(* Logix 5000 project; controller RSL5k_18_Template_noLib Emulate 5570 rev 32.11; software revision 32.02; part 2 of 16 *)
(* tags used below, declared in another part *)
   Inp_PV : REAL;   // Input Signal (process variable) from Sensor
   Inp_PVSrcQ : DINT;   // Input Source and Quality (from Channel object, if available) (enum)
   Inp_PVNotify : DINT;   // Related PV object alarm prio and ack status (enum)
   Inp_PVBad : BOOL;   // 1=PV or I/O Comms Status Bad, 0=OK
   Inp_PVUncertain : BOOL;   // 1=PV Value Not Reliable, 0=OK
   Inp_Sim : BOOL;   // 1=Use simulated PV (Set_SimPV); 0=Use Input (Inp_PV)
   Cfg_UseChanSrcQ : BOOL;   // 1=Pass thru connected Channel's SrcQ value, 0=generate SrcQ
   Cfg_FiltTC : REAL;   // PV Filter Time Constant (s), 0.0 = unfiltered
   Cfg_HiHiLim : REAL;   // High-High Status Threshold (EU)
   Cfg_HiHiDB : REAL;   // High-High Status Deadband (EU)
   Cfg_HiLim : REAL;   // High Status Threshold (EU)
   Cfg_HiDB : REAL;   // High Status Deadband (EU)
   Cfg_LoLim : REAL;   // Low Status Threshold (EU)
   Cfg_LoDB : REAL;   // Low Status Deadband (EU)
   Cfg_LoLoLim : REAL;   // Low-Low Status Threshold (EU)
   Cfg_LoLoDB : REAL;   // Low-Low Status Deadband (EU)
   Cfg_FailHiLim : REAL;   // Out-of-Range (fail) High Limit (raw units)
   Cfg_FailLoLim : REAL;   // Out-of-Range (fail) Low Limit (raw units)
   Cfg_FailDB : REAL;   // Out-of-Range (fail) High/Low Deadband (raw units)
   Set_SimPV : REAL;   // PV used in Simulation (Inp_Sim=1) (EU)
   PCmd_ClearCapt : BOOL;   // Program Command to Clear the captured min / max PV excursion values
   Val : REAL;   // Analog Value (after Substitute PV, if used)
   Val_InpPV : REAL;   // Analog Input Value (actual, before Substitute PV selection)
   Val_PVMinCapt : REAL;   // Captured PV Minimum (excursion) since last cleared
   Val_PVMaxCapt : REAL;   // Captured PV Maximum (excursion) since last cleared
   SrcQ_IO : DINT;   // Source and Quality of primary I/O (enumeration)
   SrcQ : DINT;   // Source and Quality of primary Val/Sts (enumeration)
   Val_Fault : DINT;   // Device Fault Status 0=none, 20=Lo, 21=Hi, 24=LoLo, 25=HiHi, 32=Fail, 34=CfgErr
   Val_NotifyAll : DINT;   // Highest Alarm prio and ack status this object + channel (enum)
   Val_UnackAlmC : DINT;   // Count of Unacknowledged Alarms
   Sts_SubstPV : BOOL;   // 1=Using Substitute PV (overrides input), 0=Using live Input PV from device
   Sts_PVBad : BOOL;   // 1=PV Bad quality or Out of Range
   Sts_PVUncertain : BOOL;   // 1=PV Value is Uncertain (quality)
   Sts_AlmInh : BOOL;   // 1=An Alarm is Shelved, Disabled or Suppressed: display icon
   Sts_Err : BOOL;   // 1=Error in Config (see detail Err_ bits for reason), display icon
   Err_Raw : BOOL;   // 1=Error in Config: Raw Input Scaling Min = Max
   Err_EU : BOOL;   // 1=Error in Config: Scaled EU Min = Max
   Err_Timer : BOOL;   // 1=Error in Config: On Delay, Off Delay, Gate Delay Time Invalid (use 0 to 2147483 s)
   Err_Filt : BOOL;   // 1=Error in Config: PV filter params (RateTime, TC)
   Err_Alarm : BOOL;   // 1=Error in Config: Alarm Min On Time, Shelf Time, Severity
   Sts_RdyReset : ALIAS FOR ORdy_Reset;   // 1=A latched alarm or shed condition is ready to be reset
   Sts_RdyAck : BOOL;   // 1=An alarm is ready to be acknowledged
   Sts_HiHiCmp : ALIAS FOR HiHiGate.Inp;   // PV High-High comparison result 1=High-High
   Sts_HiHi : ALIAS FOR HiHi.Inp;   // 1=Analog Input is above High-High limit
   Sts_HiCmp : ALIAS FOR HiGate.Inp;   // PV High comparison result 1=High
   Sts_Hi : ALIAS FOR Hi.Inp;   // 1=Analog Input is above High limit
   Sts_LoCmp : ALIAS FOR LoGate.Inp;   // PV Low comparison result 1=Low
   Sts_Lo : ALIAS FOR Lo.Inp;   // 1=Analog Input is below Low limit
   Sts_LoLoCmp : ALIAS FOR LoLoGate.Inp;   // PV Low-Low comparison result 1=Low-Low
   Sts_LoLo : ALIAS FOR LoLo.Inp;   // 1=Analog Input is below Low-Low limit
   Sts_FailCmp : ALIAS FOR FailGate.Inp;   // PV Fail comparison result 1=Out of Range
   Sts_Fail : ALIAS FOR Fail.Inp;   // 1=Analog Input is Out of Range or PV Bad
   P_AIn : BOOL;   // Unique Parameter Name for auto - discovery
   LoLo : P_Alarm;   // Low-Low Alarm
   Lo : P_Alarm;   // Low Alarm
   Hi : P_Alarm;   // High Alarm
   HiHi : P_Alarm;   // High-High Alarm
   Fail : P_Alarm;   // Analog Input Failure Alarm (bad quality or out of range)
   Wrk_Notify : DINT;   // Buffer for building Val_Notify
   Wrk_Fault : DINT;   // Buffer for building Val_Fault
   Wrk_SrcQ : DINT;   // Register for building Source / Quality enumeration
   Wrk_SubstPV : BOOL;   // Internal flag: Using Substitute PV
   Wrk_UnfiltPV : REAL;   // Unfiltered PV, input to 1st order filter
   Wrk_Alpha : REAL;   // Filter multiplier = (1 / (1+TC/dT) )
   Wrk_ScanT : TIMER;   // Scan Timer (milliseconds, always runs)
   Wrk_ScanTime : REAL;   // Time since this instance was last scanned
   Wrk_FiltPV : REAL;   // Filtered PV
   Wrk_ValidONS : BOOL;   // Selected PV goes from Infinite or Not a Number to VALID
   Wrk_SelPVDINT : DINT;   // Selected PV check for Infinite or Non A Number
   Wrk_SelPVInfNaN : BOOL;   // Selected PV (Input or Substitute) is Infinite or NaN
   Wrk_Fail : BOOL;   // Internal flag: Fail Status
   Wrk_LoLo : BOOL;   // Internal flag: Low-Low Status
   Wrk_Lo : BOOL;   // Internal flag: Low Status
   Wrk_Hi : BOOL;   // Internal flag: High Status
   Wrk_HiHi : BOOL;   // Internal flag: High-High Status
   FailGate : P_Gate;   // Fail Alarm Gate / Delay Block
   LoLoGate : P_Gate;   // Low-Low Alarm Gate / Delay Block
   LoGate : P_Gate;   // Low Alarm Gate / Delay Block
   HiHiGate : P_Gate;   // High-High Alarm Gate / Delay Block
   HiGate : P_Gate;   // High Alarm Gate / Delay Block
   Wrk_InpInfNaN : BOOL;   // Input is Infinite or Not a Number
   Wrk_UnackAlmC : DINT;   // Buffer for building Val_UnackAlmC
   Val_Notify : DINT;   // Highest Alarm prio and ack status this object only (enum)
   ORdy_ResetAckAll : BOOL;   // 1=Ready for OCmd_ResetAckAll (enables HMI button)
   ORdy_Reset : BOOL;   // 1=Ready for OCmd_Reset (enables HMI button)
   OCmd_ClearCapt : BOOL;   // Operator Command to Clear the captured min / max PV excursion values
   MSet_SubstPV : REAL;   // Maintenance-Entered Substitute PV (EU)
   Wrk_RawPV : REAL;   // Value of raw PV to be used for Out of Range checking
(* P_AIn, continued *)

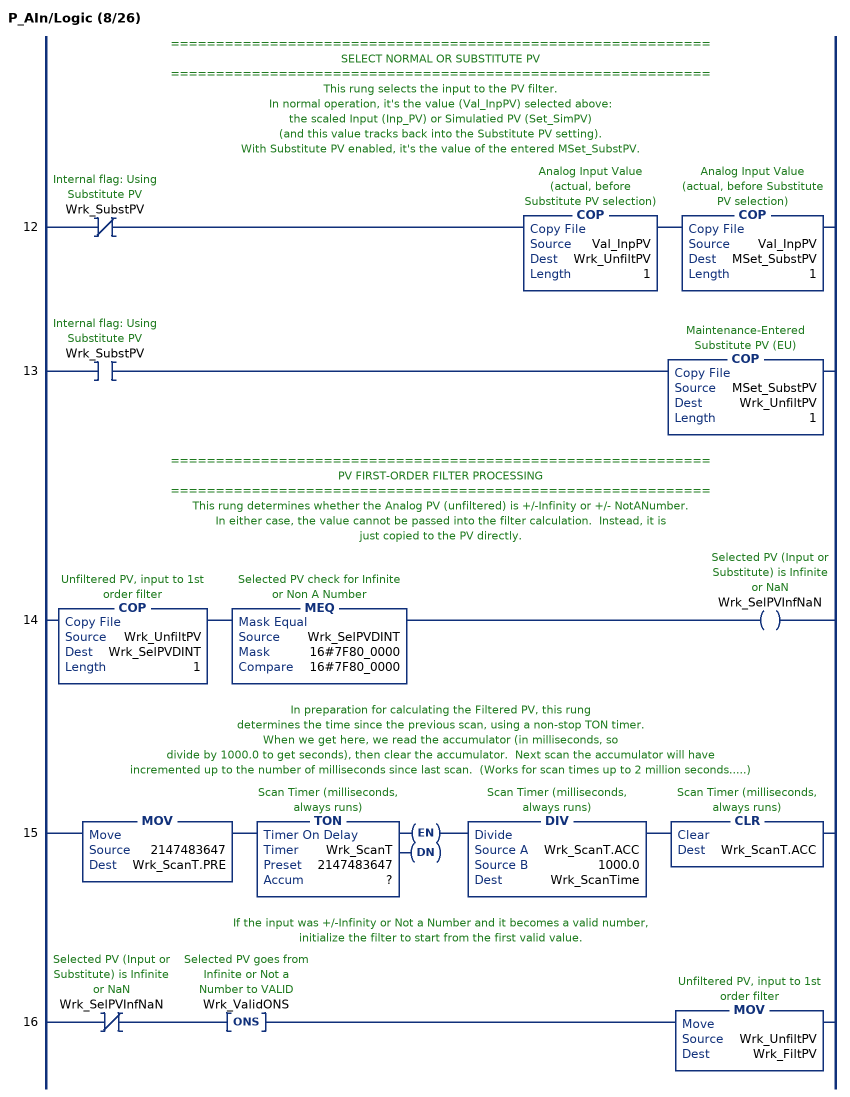
   [picture p24: P_AIn/Logic rungs 12-16]
   // ============================================================
   // SELECT NORMAL OR SUBSTITUTE PV
   // ============================================================
   // This rung selects the input to the PV filter.
   // In normal operation, it's the value (Val_InpPV) selected above:
   // the scaled Input (Inp_PV) or Simulatied PV (Set_SimPV)
   // (and this value tracks back into the Substitute PV setting).
   // With Substitute PV enabled, it's the value of the entered MSet_SubstPV.
   12: XIO(Wrk_SubstPV)COP(Val_InpPV,Wrk_UnfiltPV,1)COP(Val_InpPV,MSet_SubstPV,1);
   13: XIC(Wrk_SubstPV)COP(MSet_SubstPV,Wrk_UnfiltPV,1);
   // ============================================================
   // PV FIRST-ORDER FILTER PROCESSING
   // ============================================================
   // This rung determines whether the Analog PV (unfiltered) is +/-Infinity or +/- NotANumber.
   // In either case, the value cannot be passed into the filter calculation.  Instead, it is
   // just copied to the PV directly.
   14: COP(Wrk_UnfiltPV,Wrk_SelPVDINT,1)MEQ(Wrk_SelPVDINT,16#7F80_0000,16#7F80_0000)OTE(Wrk_SelPVInfNaN);
   // In preparation for calculating the Filtered PV, this rung
   // determines the time since the previous scan, using a non-stop TON timer.
   // When we get here, we read the accumulator (in milliseconds, so
   // divide by 1000.0 to get seconds), then clear the accumulator.  Next scan the accumulator will have
   // incremented up to the number of milliseconds since last scan.  (Works for scan times up to 2 million seconds.....)
   15: MOV(2147483647,Wrk_ScanT.PRE)TON(Wrk_ScanT,?,?)DIV(Wrk_ScanT.ACC,1000.0,Wrk_ScanTime)CLR(Wrk_ScanT.ACC);
   // If the input was +/-Infinity or Not a Number and it becomes a valid number,
   // initialize the filter to start from the first valid value.
   16: XIO(Wrk_SelPVInfNaN)ONS(Wrk_ValidONS)MOV(Wrk_UnfiltPV,Wrk_FiltPV);
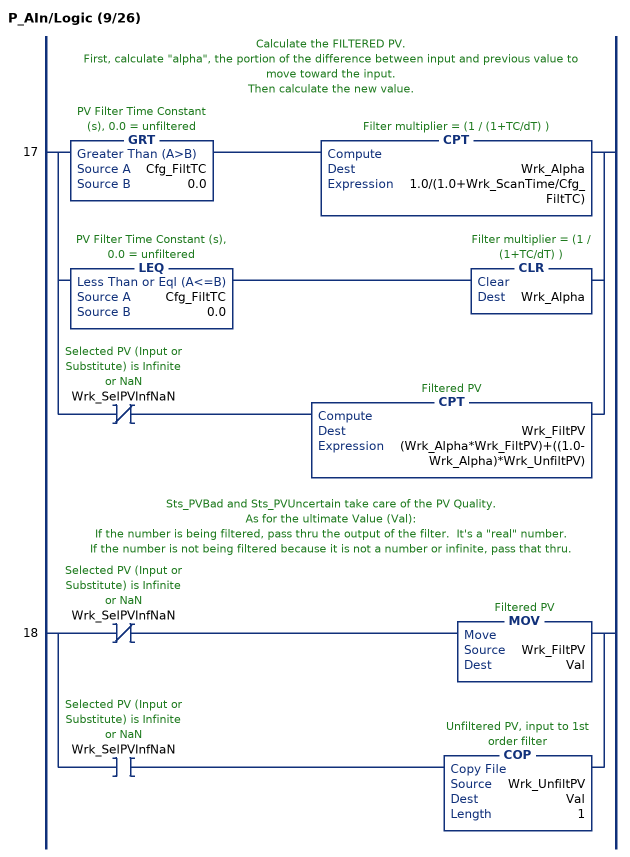
   // Calculate the FILTERED PV.
   // First, calculate "alpha", the portion of the difference between input and previous value to move toward the input.
   // Then calculate the new value.
   17: [GRT(Cfg_FiltTC,0.0) CPT(Wrk_Alpha,1.0/(1.0+Wrk_ScanTime/Cfg_FiltTC)) ,LEQ(Cfg_FiltTC,0.0) CLR(Wrk_Alpha) ,XIO(Wrk_SelPVInfNaN) CPT(Wrk_FiltPV,(Wrk_Alpha*Wrk_FiltPV)+((1.0-Wrk_Alpha)*Wrk_UnfiltPV)) ];
   // Sts_PVBad and Sts_PVUncertain take care of the PV Quality.
   // As for the ultimate Value (Val):
   // If the number is being filtered, pass thru the output of the filter.  It's a "real" number.
   // If the number is not being filtered because it is not a number or infinite, pass that thru.
   18: [XIO(Wrk_SelPVInfNaN) MOV(Wrk_FiltPV,Val) ,XIC(Wrk_SelPVInfNaN) COP(Wrk_UnfiltPV,Val,1) ];
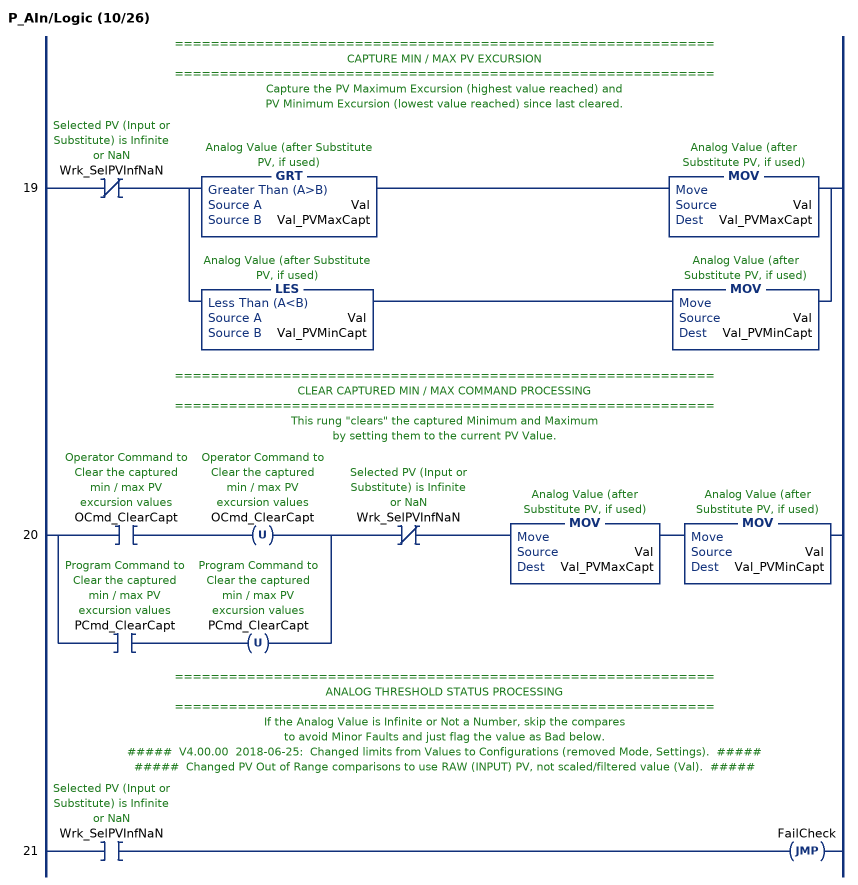
   // ============================================================
   // CAPTURE MIN / MAX PV EXCURSION
   // ============================================================
   // Capture the PV Maximum Excursion (highest value reached) and
   // PV Minimum Excursion (lowest value reached) since last cleared.
   19: XIO(Wrk_SelPVInfNaN)[GRT(Val,Val_PVMaxCapt) MOV(Val,Val_PVMaxCapt) ,LES(Val,Val_PVMinCapt) MOV(Val,Val_PVMinCapt) ];
   // ============================================================
   // CLEAR CAPTURED MIN / MAX COMMAND PROCESSING
   // ============================================================
   // This rung "clears" the captured Minimum and Maximum
   // by setting them to the current PV Value.
   20: [XIC(OCmd_ClearCapt) OTU(OCmd_ClearCapt) ,XIC(PCmd_ClearCapt) OTU(PCmd_ClearCapt) ]XIO(Wrk_SelPVInfNaN)MOV(Val,Val_PVMaxCapt)MOV(Val,Val_PVMinCapt);
   // ============================================================
   // ANALOG THRESHOLD STATUS PROCESSING
   // ============================================================
   // If the Analog Value is Infinite or Not a Number, skip the compares
   // to avoid Minor Faults and just flag the value as Bad below.
   // #####  V4.00.00  2018-06-25:  Changed limits from Values to Configurations (removed Mode, Settings).  #####
   // #####  Changed PV Out of Range comparisons to use RAW (INPUT) PV, not scaled/filtered value (Val).  #####
   21: XIC(Wrk_SelPVInfNaN)JMP(FailCheck);
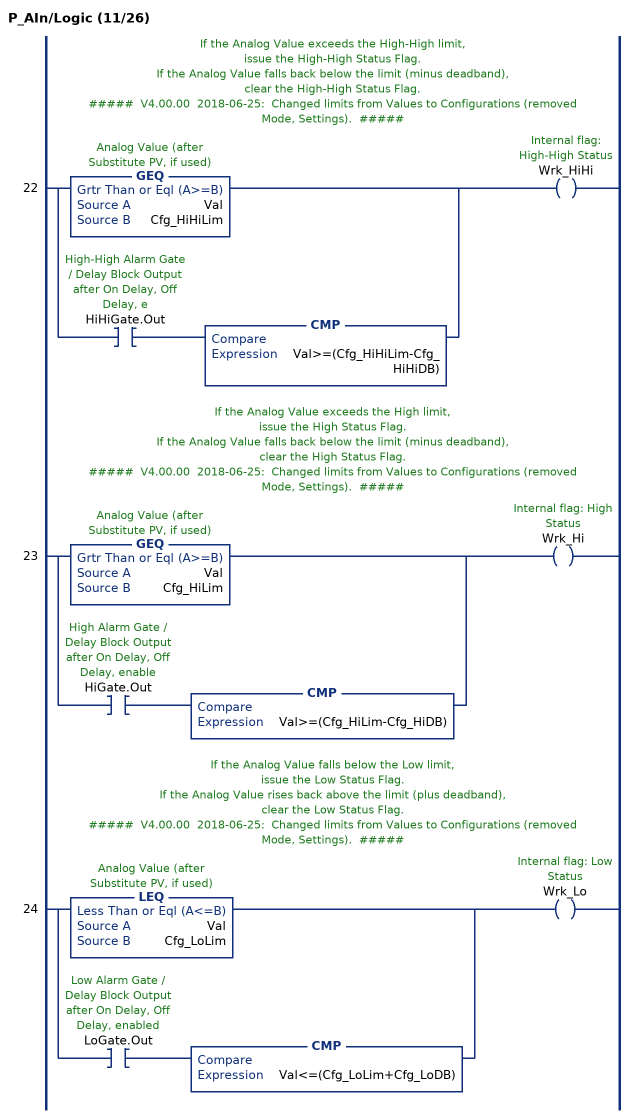
   // If the Analog Value exceeds the High-High limit,
   // issue the High-High Status Flag.
   // If the Analog Value falls back below the limit (minus deadband),
   // clear the High-High Status Flag.
   // #####  V4.00.00  2018-06-25:  Changed limits from Values to Configurations (removed Mode, Settings).  #####
   22: [GEQ(Val,Cfg_HiHiLim) ,XIC(HiHiGate.Out) CMP(Val>=(Cfg_HiHiLim-Cfg_HiHiDB)) ]OTE(Wrk_HiHi);
   // If the Analog Value exceeds the High limit,
   // issue the High Status Flag.
   // If the Analog Value falls back below the limit (minus deadband),
   // clear the High Status Flag.
   // #####  V4.00.00  2018-06-25:  Changed limits from Values to Configurations (removed Mode, Settings).  #####
   23: [GEQ(Val,Cfg_HiLim) ,XIC(HiGate.Out) CMP(Val>=(Cfg_HiLim-Cfg_HiDB)) ]OTE(Wrk_Hi);
   // If the Analog Value falls below the Low limit,
   // issue the Low Status Flag.
   // If the Analog Value rises back above the limit (plus deadband),
   // clear the Low Status Flag.
   // #####  V4.00.00  2018-06-25:  Changed limits from Values to Configurations (removed Mode, Settings).  #####
   24: [LEQ(Val,Cfg_LoLim) ,XIC(LoGate.Out) CMP(Val<=(Cfg_LoLim+Cfg_LoDB)) ]OTE(Wrk_Lo);
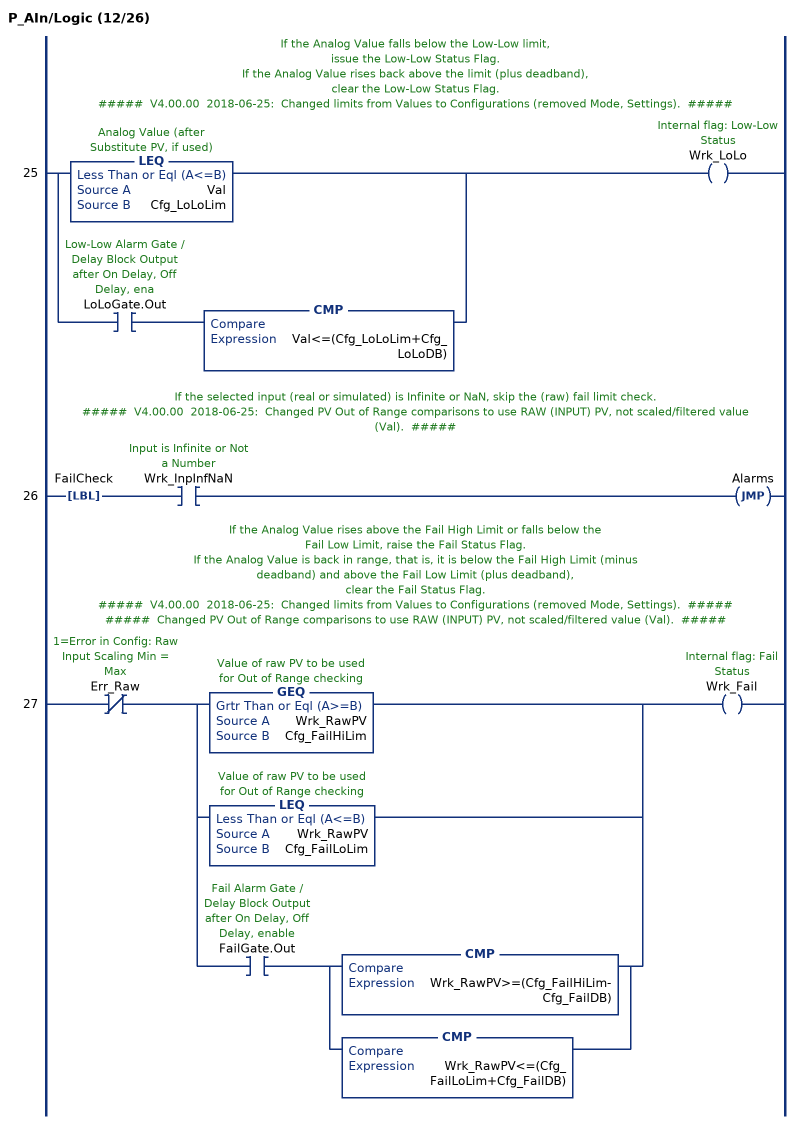
   // If the Analog Value falls below the Low-Low limit,
   // issue the Low-Low Status Flag.
   // If the Analog Value rises back above the limit (plus deadband),
   // clear the Low-Low Status Flag.
   // #####  V4.00.00  2018-06-25:  Changed limits from Values to Configurations (removed Mode, Settings).  #####
   25: [LEQ(Val,Cfg_LoLoLim) ,XIC(LoLoGate.Out) CMP(Val<=(Cfg_LoLoLim+Cfg_LoLoDB)) ]OTE(Wrk_LoLo);
   // If the selected input (real or simulated) is Infinite or NaN, skip the (raw) fail limit check.
   // #####  V4.00.00  2018-06-25:  Changed PV Out of Range comparisons to use RAW (INPUT) PV, not scaled/filtered value (Val).  #####
   26: LBL(FailCheck)XIC(Wrk_InpInfNaN)JMP(Alarms);
   // If the Analog Value rises above the Fail High Limit or falls below the
   // Fail Low Limit, raise the Fail Status Flag.
   // If the Analog Value is back in range, that is, it is below the Fail High Limit (minus
   // deadband) and above the Fail Low Limit (plus deadband),
   // clear the Fail Status Flag.
   // #####  V4.00.00  2018-06-25:  Changed limits from Values to Configurations (removed Mode, Settings).  #####
   // #####  Changed PV Out of Range comparisons to use RAW (INPUT) PV, not scaled/filtered value (Val).  #####
   27: XIO(Err_Raw)[[GEQ(Wrk_RawPV,Cfg_FailHiLim) ,LEQ(Wrk_RawPV,Cfg_FailLoLim) ] ,XIC(FailGate.Out) [CMP(Wrk_RawPV>=(Cfg_FailHiLim-Cfg_FailDB)) ,CMP(Wrk_RawPV<=(Cfg_FailLoLim+Cfg_FailDB)) ] ]OTE(Wrk_Fail);
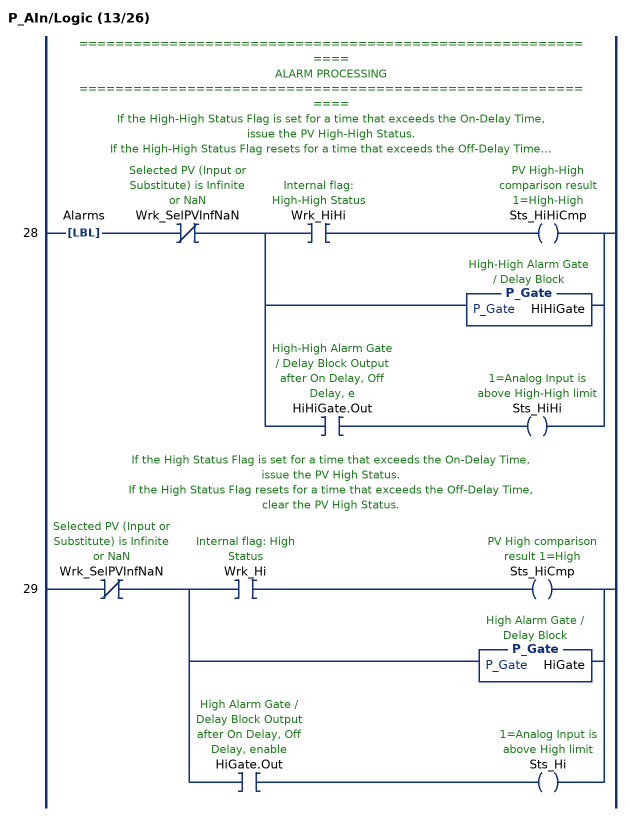
   // ============================================================
   // ALARM PROCESSING
   // ============================================================
   // If the High-High Status Flag is set for a time that exceeds the On-Delay Time,
   // issue the PV High-High Status.
   // If the High-High Status Flag resets for a time that exceeds the Off-Delay Time,
   // clear the PV High-High Status.
   28: LBL(Alarms)XIO(Wrk_SelPVInfNaN)[XIC(Wrk_HiHi) OTE(Sts_HiHiCmp) ,P_Gate(HiHiGate) ,XIC(HiHiGate.Out) OTE(Sts_HiHi) ];
   // If the High Status Flag is set for a time that exceeds the On-Delay Time,
   // issue the PV High Status.
   // If the High Status Flag resets for a time that exceeds the Off-Delay Time,
   // clear the PV High Status.
   29: XIO(Wrk_SelPVInfNaN)[XIC(Wrk_Hi) OTE(Sts_HiCmp) ,P_Gate(HiGate) ,XIC(HiGate.Out) OTE(Sts_Hi) ];
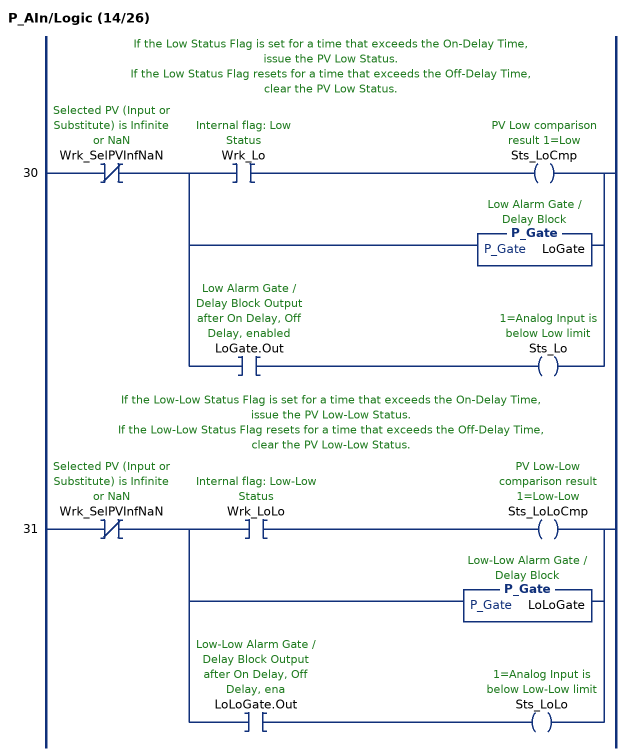
   // If the Low Status Flag is set for a time that exceeds the On-Delay Time,
   // issue the PV Low Status.
   // If the Low Status Flag resets for a time that exceeds the Off-Delay Time,
   // clear the PV Low Status.
   30: XIO(Wrk_SelPVInfNaN)[XIC(Wrk_Lo) OTE(Sts_LoCmp) ,P_Gate(LoGate) ,XIC(LoGate.Out) OTE(Sts_Lo) ];
   // If the Low-Low Status Flag is set for a time that exceeds the On-Delay Time,
   // issue the PV Low-Low Status.
   // If the Low-Low Status Flag resets for a time that exceeds the Off-Delay Time,
   // clear the PV Low-Low Status.
   31: XIO(Wrk_SelPVInfNaN)[XIC(Wrk_LoLo) OTE(Sts_LoLoCmp) ,P_Gate(LoLoGate) ,XIC(LoLoGate.Out) OTE(Sts_LoLo) ];
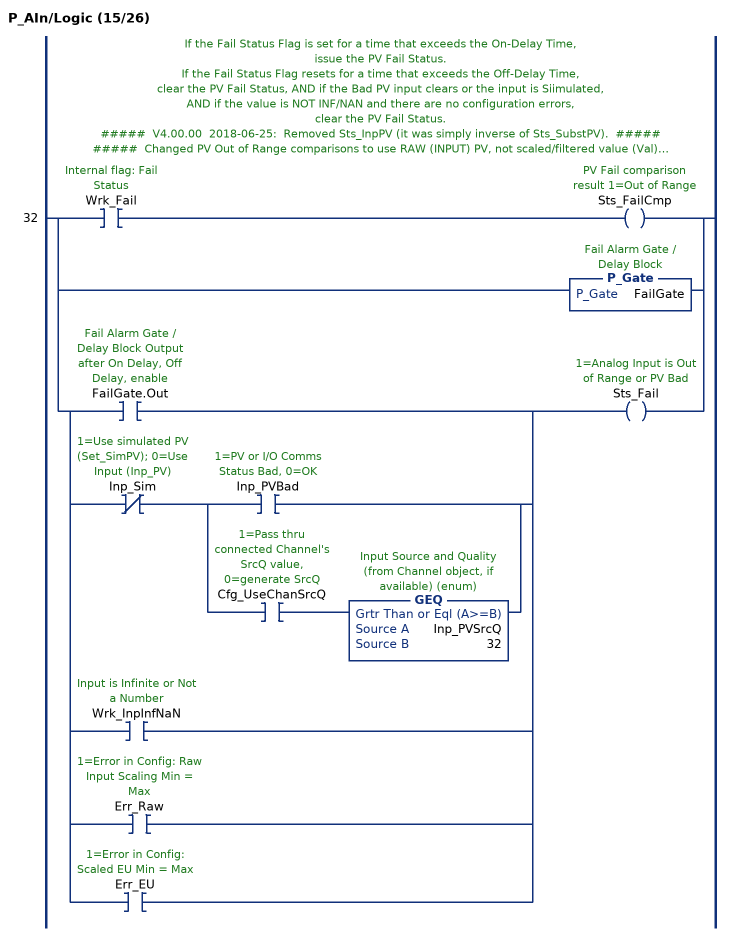
   // If the Fail Status Flag is set for a time that exceeds the On-Delay Time,
   // issue the PV Fail Status.
   // If the Fail Status Flag resets for a time that exceeds the Off-Delay Time,
   // clear the PV Fail Status, AND if the Bad PV input clears or the input is Siimulated,
   // AND if the value is NOT INF/NAN and there are no configuration errors,
   // clear the PV Fail Status.
   // #####  V4.00.00  2018-06-25:  Removed Sts_InpPV (it was simply inverse of Sts_SubstPV).  #####
   // #####  Changed PV Out of Range comparisons to use RAW (INPUT) PV, not scaled/filtered value (Val).  #####
   32: [XIC(Wrk_Fail) OTE(Sts_FailCmp) ,P_Gate(FailGate) ,[XIC(FailGate.Out) ,XIO(Inp_Sim) [XIC(Inp_PVBad) ,XIC(Cfg_UseChanSrcQ) GEQ(Inp_PVSrcQ,32) ] ,XIC(Wrk_InpInfNaN) ,XIC(Err_Raw) ,XIC(Err_EU) ] OTE(Sts_Fail) ];
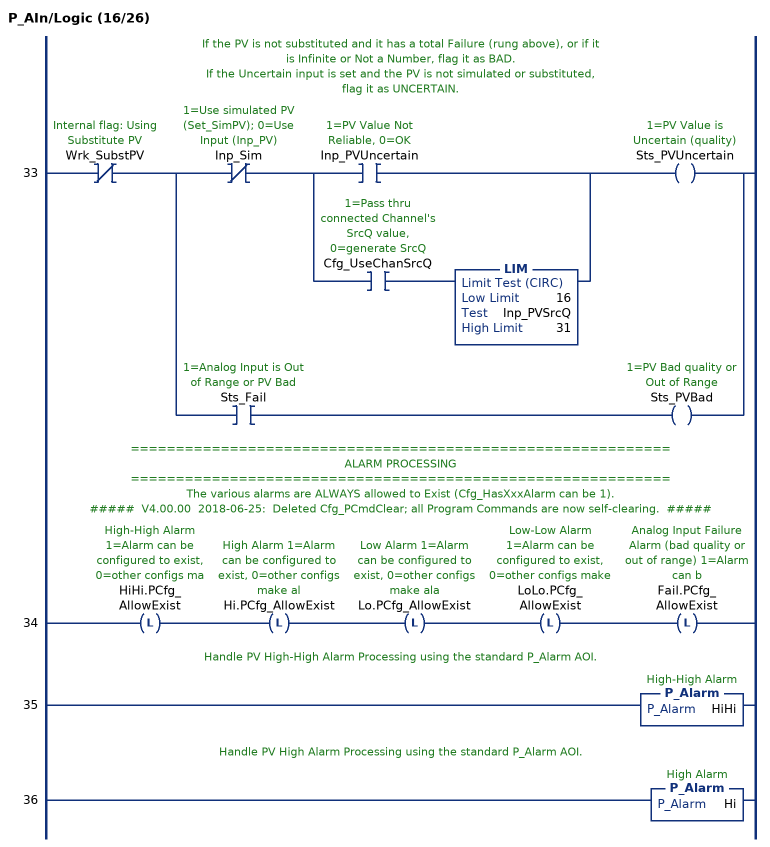
   // If the PV is not substituted and it has a total Failure (rung above), or if it
   // is Infinite or Not a Number, flag it as BAD.
   // If the Uncertain input is set and the PV is not simulated or substituted,
   // flag it as UNCERTAIN.
   33: XIO(Wrk_SubstPV)[XIO(Inp_Sim) [XIC(Inp_PVUncertain) ,XIC(Cfg_UseChanSrcQ) LIM(16,Inp_PVSrcQ,31) ] OTE(Sts_PVUncertain) ,XIC(Sts_Fail) OTE(Sts_PVBad) ];
   // ============================================================
   // ALARM PROCESSING
   // ============================================================
   // The various alarms are ALWAYS allowed to Exist (Cfg_HasXxxAlarm can be 1).
   // #####  V4.00.00  2018-06-25:  Deleted Cfg_PCmdClear; all Program Commands are now self-clearing.  #####
   34: OTL(HiHi.PCfg_AllowExist)OTL(Hi.PCfg_AllowExist)OTL(Lo.PCfg_AllowExist)OTL(LoLo.PCfg_AllowExist)OTL(Fail.PCfg_AllowExist);
   // Handle PV High-High Alarm Processing using the standard P_Alarm AOI.
   35: P_Alarm(HiHi);
   // Handle PV High Alarm Processing using the standard P_Alarm AOI.
   36: P_Alarm(Hi);
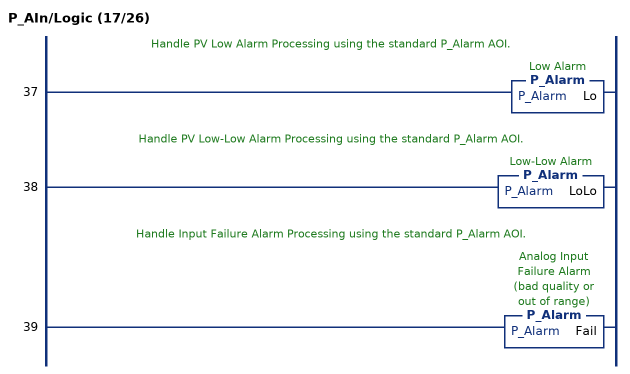
   // Handle PV Low Alarm Processing using the standard P_Alarm AOI.
   37: P_Alarm(Lo);
   // Handle PV Low-Low Alarm Processing using the standard P_Alarm AOI.
   38: P_Alarm(LoLo);
   // Handle Input Failure Alarm Processing using the standard P_Alarm AOI.
   39: P_Alarm(Fail);
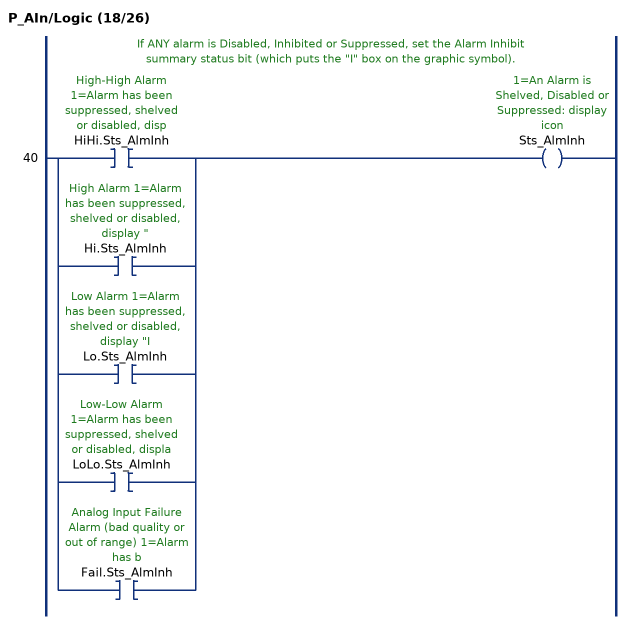
   // If ANY alarm is Disabled, Inhibited or Suppressed, set the Alarm Inhibit
   // summary status bit (which puts the "I" box on the graphic symbol).
   40: [XIC(HiHi.Sts_AlmInh) ,XIC(Hi.Sts_AlmInh) ,XIC(Lo.Sts_AlmInh) ,XIC(LoLo.Sts_AlmInh) ,XIC(Fail.Sts_AlmInh) ]OTE(Sts_AlmInh);
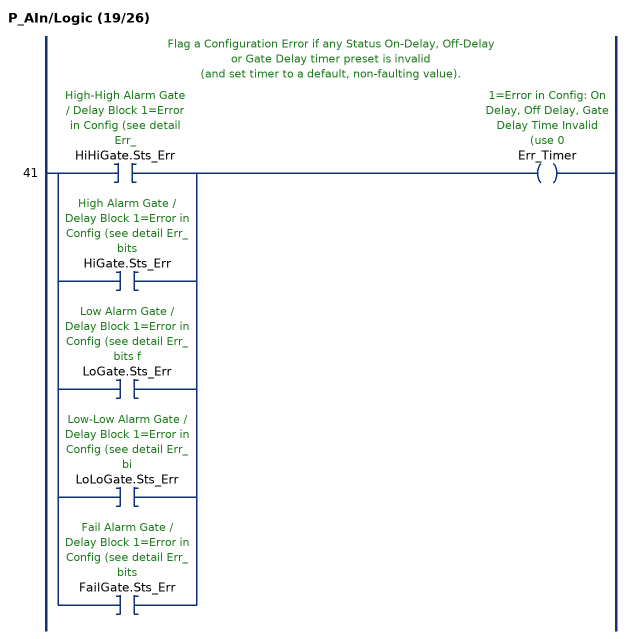
   // Flag a Configuration Error if any Status On-Delay, Off-Delay
   // or Gate Delay timer preset is invalid
   // (and set timer to a default, non-faulting value).
   41: [XIC(HiHiGate.Sts_Err) ,XIC(HiGate.Sts_Err) ,XIC(LoGate.Sts_Err) ,XIC(LoLoGate.Sts_Err) ,XIC(FailGate.Sts_Err) ]OTE(Err_Timer);
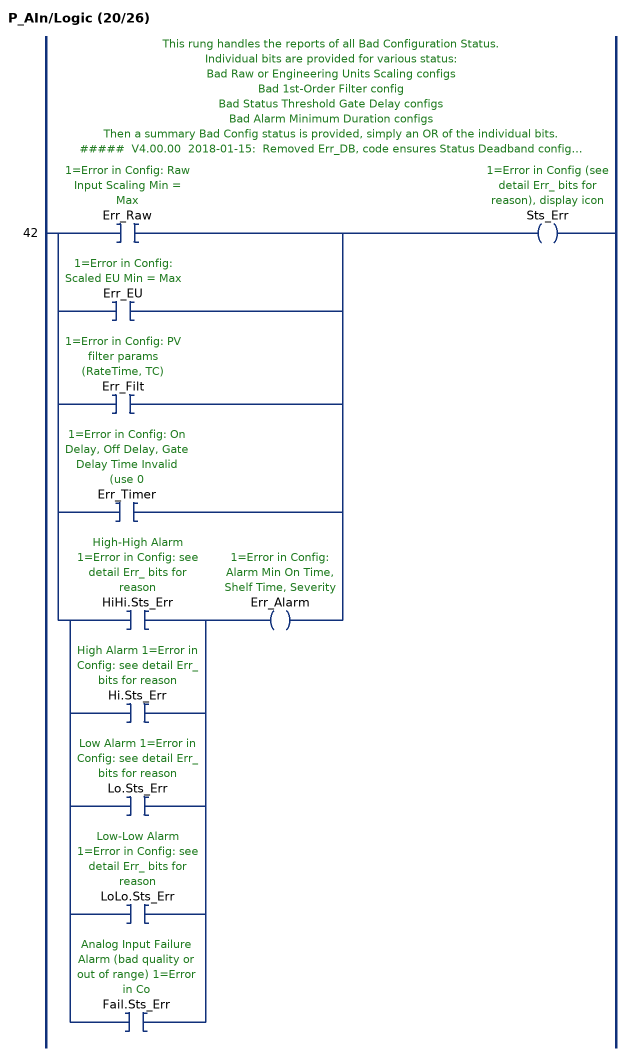
   // This rung handles the reports of all Bad Configuration Status.
   // Individual bits are provided for various status:
   // Bad Raw or Engineering Units Scaling configs
   // Bad 1st-Order Filter config
   // Bad Status Threshold Gate Delay configs
   // Bad Alarm Minimum Duration configs
   // Then a summary Bad Config status is provided, simply an OR of the individual bits.
   // #####  V4.00.00  2018-01-15:  Removed Err_DB, code ensures Status Deadband configs are always valid.  #####
   42: [XIC(Err_Raw) ,XIC(Err_EU) ,XIC(Err_Filt) ,XIC(Err_Timer) ,[XIC(HiHi.Sts_Err) ,XIC(Hi.Sts_Err) ,XIC(Lo.Sts_Err) ,XIC(LoLo.Sts_Err) ,XIC(Fail.Sts_Err) ] OTE(Err_Alarm) ]OTE(Sts_Err);
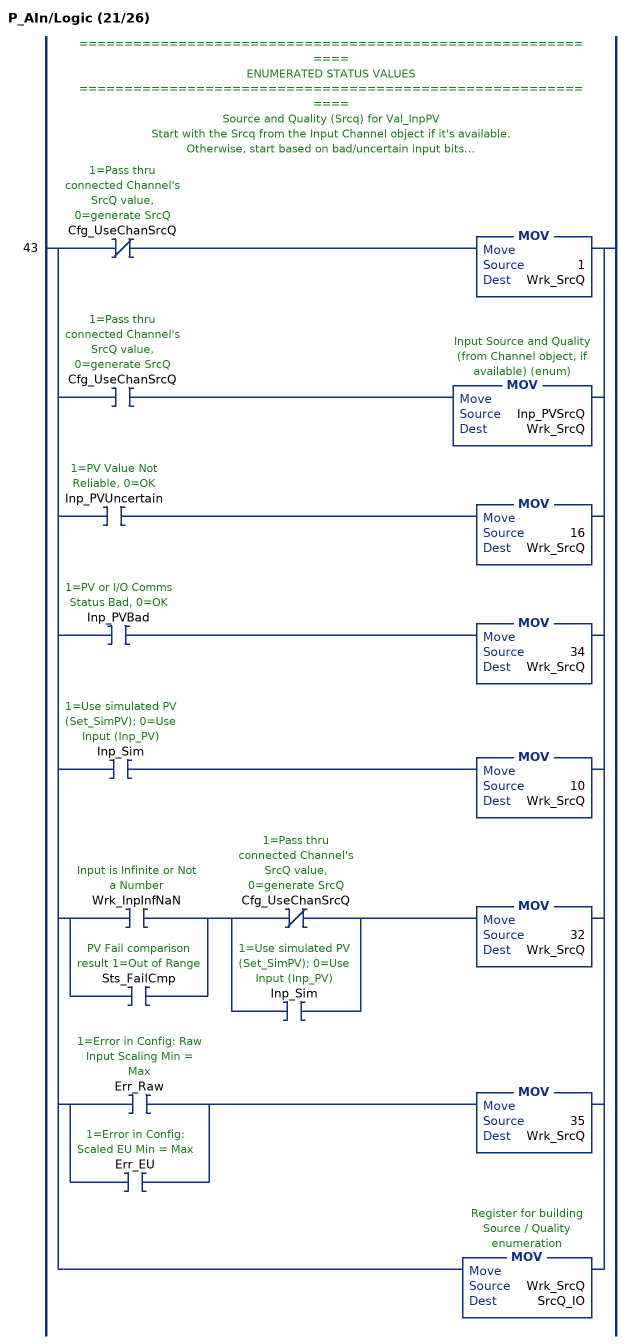
   // ============================================================
   // ENUMERATED STATUS VALUES
   // ============================================================
   // Source and Quality (Srcq) for Val_InpPV
   // Start with the Srcq from the Input Channel object if it's available.
   // Otherwise, start based on bad/uncertain input bits.
   // 0 = Good: live, confirmed good;   1 = Good: live, assumed good;
   // 2 = Good: no feedback, assumed good;   8 = Test: Simulated;   9 = Test: Loopback;
   // 10 = Test: Manually Entered;   16 = Uncertain: Live, off-spec;
   // 17 = Uncertain, Substituted at Device / Bus;   18 = Uncertain, Substituted at AOI;
   // 19 = Uncertain, using last known good;    20 = Uncertain, using replacement value;
   // 32 = Bad, Signal Failure;   33 = Bad, Channel Fault;
   // 34 = Bad, Module / Comms Fault;   35 = Bad, Invalid Configuration
   // #####  V4.00.00  2018-06-25:  Modified to correct precedence and value of Simulated PV.  #####
   // #####  V4.00.01  2018-08-29:  Modified handling of Simulated PV and scaling config errors.  #####
   43: [XIO(Cfg_UseChanSrcQ) MOV(1,Wrk_SrcQ) ,XIC(Cfg_UseChanSrcQ) MOV(Inp_PVSrcQ,Wrk_SrcQ) ,XIC(Inp_PVUncertain) MOV(16,Wrk_SrcQ) ,XIC(Inp_PVBad) MOV(34,Wrk_SrcQ) ,XIC(Inp_Sim) MOV(10,Wrk_SrcQ) ,[XIC(Wrk_InpInfNaN) ,XIC(Sts_FailCmp) ] [XIO(Cfg_UseChanSrcQ) ,XIC(Inp_Sim) ] MOV(32,Wrk_SrcQ) ,[XIC(Err_Raw) ,XIC(Err_EU) ] MOV(35,Wrk_SrcQ) ,MOV(Wrk_SrcQ,SrcQ_IO) ];
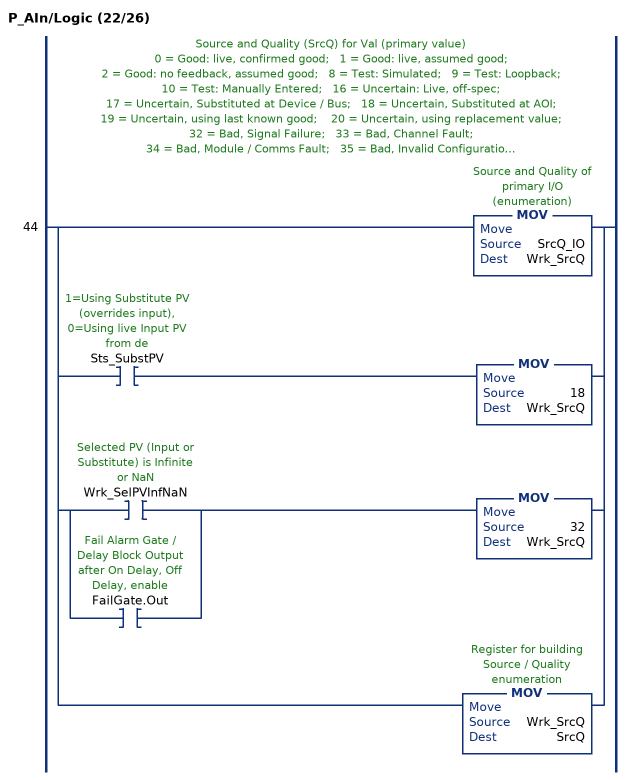
   // Source and Quality (SrcQ) for Val (primary value)
   // 0 = Good: live, confirmed good;   1 = Good: live, assumed good;
   // 2 = Good: no feedback, assumed good;   8 = Test: Simulated;   9 = Test: Loopback;
   // 10 = Test: Manually Entered;   16 = Uncertain: Live, off-spec;
   // 17 = Uncertain, Substituted at Device / Bus;   18 = Uncertain, Substituted at AOI;
   // 19 = Uncertain, using last known good;    20 = Uncertain, using replacement value;
   // 32 = Bad, Signal Failure;   33 = Bad, Channel Fault;
   // 34 = Bad, Module / Comms Fault;   35 = Bad, Invalid Configuration
   // #####  V4.00.00  2018-06-25:  Modified to allow Substitute PV to control SrcQ despite alarm for failed PV.  #####
   // #####  V4.00.01  2018-08-29:  Modified handling of Substitute PV and Channel SrcQ.  #####
   44: [MOV(SrcQ_IO,Wrk_SrcQ) ,XIC(Sts_SubstPV) MOV(18,Wrk_SrcQ) ,[XIC(Wrk_SelPVInfNaN) ,XIC(FailGate.Out) ] MOV(32,Wrk_SrcQ) ,MOV(Wrk_SrcQ,SrcQ) ];
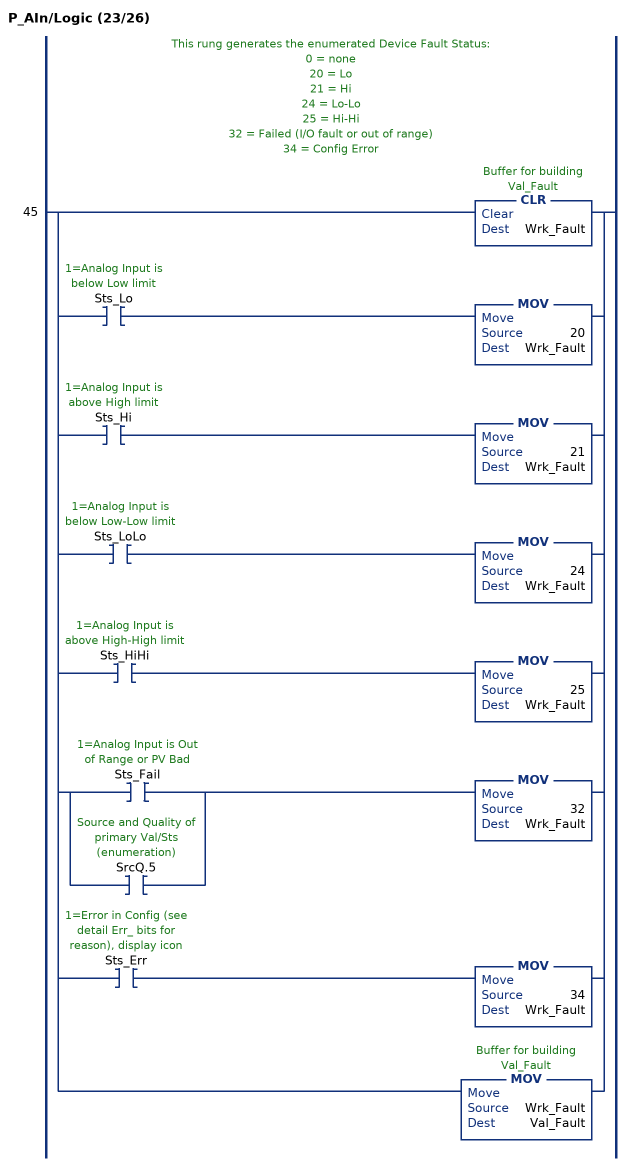
   // This rung generates the enumerated Device Fault Status:
   // 0 = none
   // 20 = Lo
   // 21 = Hi
   // 24 = Lo-Lo
   // 25 = Hi-Hi
   // 32 = Failed (I/O fault or out of range)
   // 34 = Config Error
   45: [CLR(Wrk_Fault) ,XIC(Sts_Lo) MOV(20,Wrk_Fault) ,XIC(Sts_Hi) MOV(21,Wrk_Fault) ,XIC(Sts_LoLo) MOV(24,Wrk_Fault) ,XIC(Sts_HiHi) MOV(25,Wrk_Fault) ,[XIC(Sts_Fail) ,XIC(SrcQ.5) ] MOV(32,Wrk_Fault) ,XIC(Sts_Err) MOV(34,Wrk_Fault) ,MOV(Wrk_Fault,Val_Fault) ];
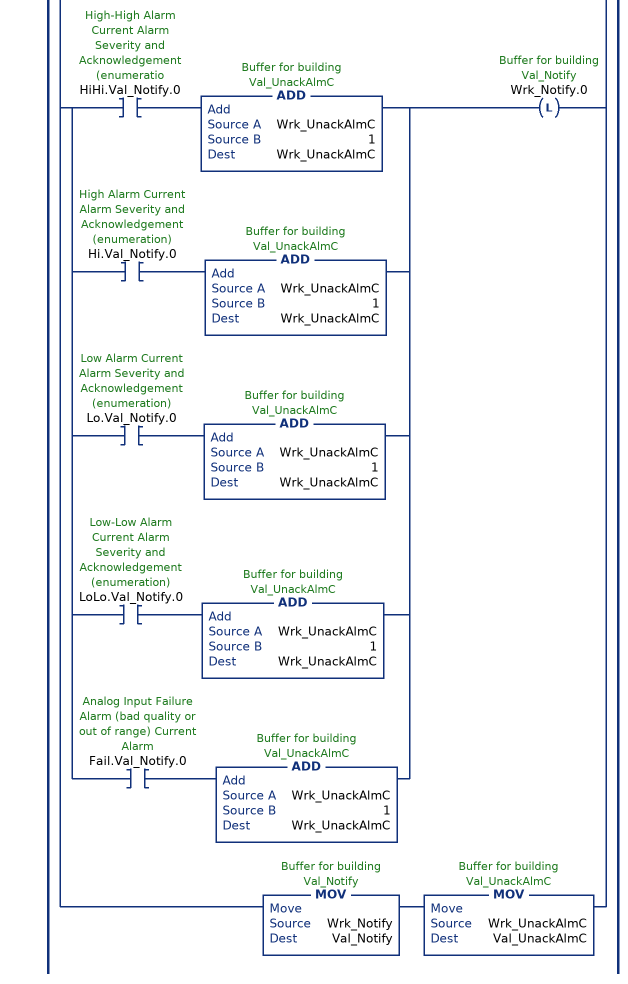
   // ============================================================
   // NOTIFICATION VALUE
   // ============================================================
   // Indicate the current alarm notification level as the max of any of the alarms,
   // and set the low-order bit for reset or ack required:
   // 0 = Not in alarm, acknowledged
   // 1 = Not in alarm, unacknowledged or reset required
   // 2 = Low severity alarm, acknowledged
   // 3 = Low severity alarm, unacknowledged
   // 4 = Medium severity alarm, acknowledged
   // 5 = Medium severity alarm, unacknowledged
   // 6 = High severity alarm, acknowledged
   // 7 = High severity alarm, unacknowledged
   // 8 = Urgent severity alarm, acknowledged
   // 9 = Urgent severity alarm, unacknowledged
   // #####  V4.00.00  2018-06-25:  Added Val_NotifyAll and Val_UnackAlmC to roll up alarm  #####
   // #####  priority / ack status and unack. alarm count including attached Channel object.  #####
   46: [CLR(Wrk_Notify) CLR(Wrk_UnackAlmC) OTU(Wrk_Notify.0) ,GRT(HiHi.Val_Notify,Wrk_Notify) MOV(HiHi.Val_Notify,Wrk_Notify) ,GRT(Hi.Val_Notify,Wrk_Notify) MOV(Hi.Val_Notify,Wrk_Notify) ,GRT(Lo.Val_Notify,Wrk_Notify) MOV(Lo.Val_Notify,Wrk_Notify) ,GRT(LoLo.Val_Notify,Wrk_Notify) MOV(LoLo.Val_Notify,Wrk_Notify) ,GRT(Fail.Val_Notify,Wrk_Notify) MOV(Fail.Val_Notify,Wrk_Notify) ,[XIC(HiHi.Val_Notify.0) ADD(Wrk_UnackAlmC,1,Wrk_UnackAlmC) ,XIC(Hi.Val_Notify.0) ADD(Wrk_UnackAlmC,1,Wrk_UnackAlmC) ,XIC(Lo.Val_Notify.0) ADD(Wrk_UnackAlmC,1,Wrk_UnackAlmC) ,XIC(LoLo.Val_Notify.0) ADD(Wrk_UnackAlmC,1,Wrk_UnackAlmC) ,XIC(Fail.Val_Notify.0) ADD(Wrk_UnackAlmC,1,Wrk_UnackAlmC) ] OTL(Wrk_Notify.0) ,MOV(Wrk_Notify,Val_Notify) MOV(Wrk_UnackAlmC,Val_UnackAlmC) ];
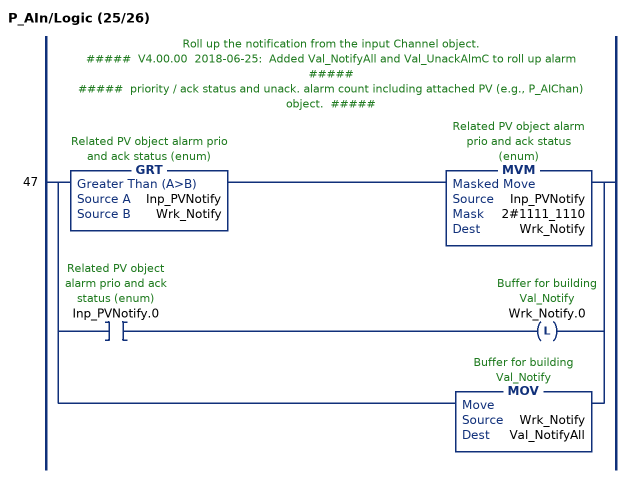
   // Roll up the notification from the input Channel object.
   // #####  V4.00.00  2018-06-25:  Added Val_NotifyAll and Val_UnackAlmC to roll up alarm  #####
   // #####  priority / ack status and unack. alarm count including attached PV (e.g., P_AIChan) object.  #####
   47: [GRT(Inp_PVNotify,Wrk_Notify) MVM(Inp_PVNotify,2#1111_1110,Wrk_Notify) ,XIC(Inp_PVNotify.0) OTL(Wrk_Notify.0) ,MOV(Wrk_Notify,Val_NotifyAll) ];
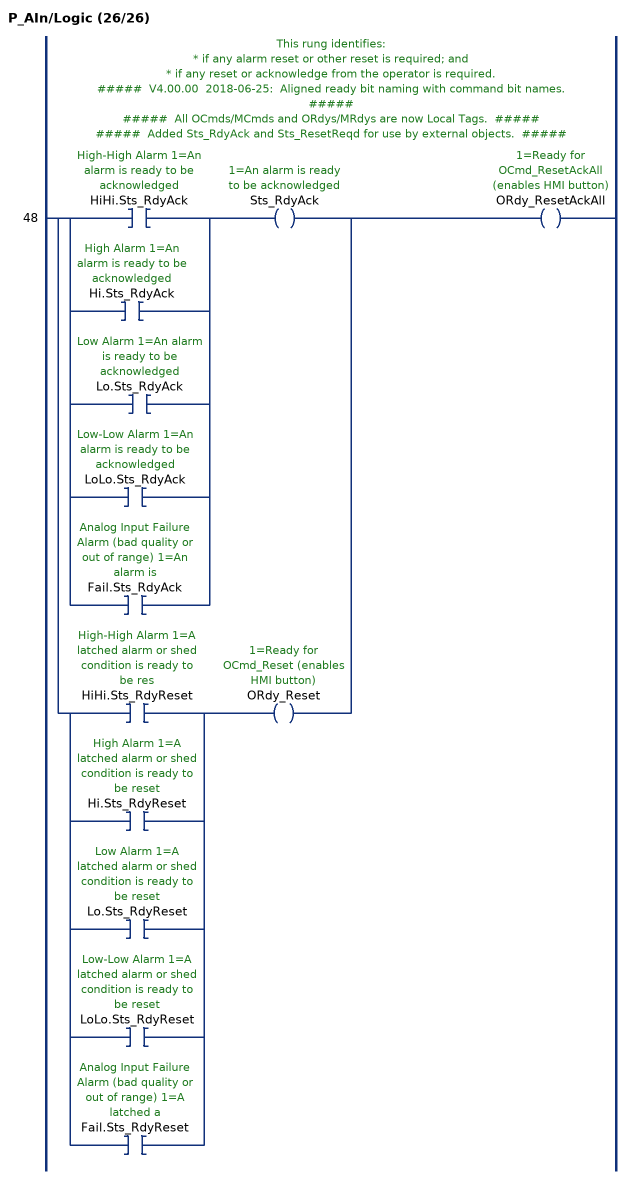
   // This rung identifies:
   // * if any alarm reset or other reset is required; and
   // * if any reset or acknowledge from the operator is required.
   // #####  V4.00.00  2018-06-25:  Aligned ready bit naming with command bit names.  #####
   // #####  All OCmds/MCmds and ORdys/MRdys are now Local Tags.  #####
   // #####  Added Sts_RdyAck and Sts_ResetReqd for use by external objects.  #####
   48: [[XIC(HiHi.Sts_RdyAck) ,XIC(Hi.Sts_RdyAck) ,XIC(Lo.Sts_RdyAck) ,XIC(LoLo.Sts_RdyAck) ,XIC(Fail.Sts_RdyAck) ] OTE(Sts_RdyAck) ,[XIC(HiHi.Sts_RdyReset) ,XIC(Hi.Sts_RdyReset) ,XIC(Lo.Sts_RdyReset) ,XIC(LoLo.Sts_RdyReset) ,XIC(Fail.Sts_RdyReset) ] OTE(ORdy_Reset) ]OTE(ORdy_ResetAckAll);
END_ROUTINE
